Staubli VAL3: pop.pgx

public program pop(MotionBuffer& x_cmd, bool& x_res)
begin
  if (nElems > 0)
    x_cmd = buffer[nPop]
    nElems = nElems - 1
    nPop = nPop + 1
    if (nPop >= size(buffer))
      nPop = 0
    endIf
    x_res = true
  else
    x_res = false
  endIf
end
